(* Logix 5000 project; controller TestController vendor 1 type 14 code 166 rev 32.11; software revision 32.02 *)
// This is a test project

TASK Continuous (continuous, watchdog 500 ms) : MainProgram   // Test continuous task
TASK EventTask (event, rate 10 ms, priority 10, watchdog 500 ms) : EventProgram01   // TestEvent Task
TASK TestTask (periodic, rate 10 ms, priority 10, watchdog 500 ms) : EquipmentPhaseProgram

MODULES
   Local : vendor 1 type 14 code 166 (ICP 0, rev 32.11)
END_MODULES

TYPE AlarmType :   // This is a test alarm type
STRUCT
   DigitalMember : CAM;   // Test digital member
END_STRUCT
END_TYPE

TYPE BoolTest :   // This is a test
STRUCT
   Member01 : BOOL;
   Member02 : BOOL;
   Member04 : BOOL;
   Member05 : BOOL;
END_STRUCT
END_TYPE

TYPE MyStringType :   // This is a test string type
STRUCT
   LEN : DINT;
   DATA : SINT[100];
END_STRUCT
END_TYPE

ADD_ON_INSTRUCTION aoi_Test   (* revision 1.0 *)
// Test AOI
VAR_INPUT
   InputTest : BOOL; {visible}
END_VAR
VAR_OUTPUT
   OutputTest : DINT; {access Read Only, visible}
END_VAR
VAR_IN_OUT
   InOutTest : SimpleType; {constant, required}
END_VAR
VAR_INPUT
   Config : INT; {access None, required}
   Test : BOOL; {access None}
END_VAR
VAR
   LocalBool : BOOL; {access None}
END_VAR

ROUTINE Logic   (* ladder *)
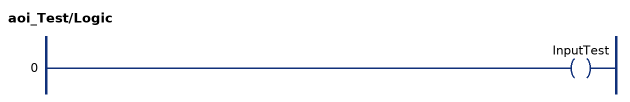
   0: OTE(InputTest);
END_ROUTINE
END_ADD_ON_INSTRUCTION

VAR_GLOBAL   (* controller tags *)
   EquipmentPhaseProgram : PHASE;
   SimpleArray : DINT[10]; {access Read Only}   // This is a test
   SimpleBool : BOOL := 1; {access None}
   SimpleDint : DINT := 3; {access None}
   SimpleInt : INT := 20; {access None}
   SimpleLint : LINT := 3; {access None}
   SimpleReal : REAL; {access None}
   SimpleSint : SINT := 20; {access None}
        .0   // This is a test
   TagParameter : SimpleType; {access None}
   TestAlarmTag : ALARM; {access None}
   TestAnalogAlarm : ALARM_ANALOG;
   TestArrayTypeTag : ArrayType; {access Read Only}
        .SintArray   // Override
   TestComplexTag : ComplexType; {access None}
   TestDigitalAlarm : ALARM_DIGITAL;
   TestStringTag : MyStringType; {access None}
   TestTag01 : SimpleType := (IntMember := 14, DintMember := 1); {access Read Only}
   TestTimer : TIMER := (PRE := 1000); {access None}   // Test Timer
END_VAR

PROGRAM EquipmentPhaseProgram
// Test

ROUTINE Resetting   (* ladder *)
   0: ;
END_ROUTINE

ROUTINE Running   (* ladder *)
END_ROUTINE
END_PROGRAM

PROGRAM EventProgram01   (* main routine Main *)

ROUTINE Main   (* ladder *)
END_ROUTINE
END_PROGRAM

PROGRAM MainProgram   (* main routine Main *)

ROUTINE FBD   (* function block diagram *)
   SHEET 1
END_ROUTINE

ROUTINE Main   (* ladder *)
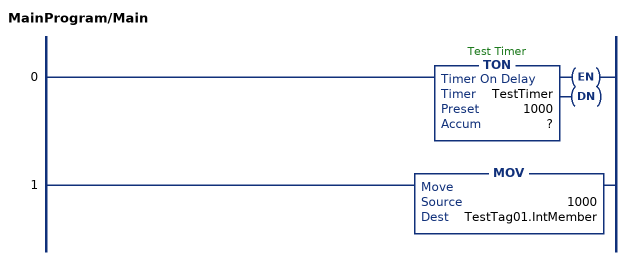
   0: TON(TestTimer,?,?);
   1: MOV(1000,TestTag01.IntMember);
END_ROUTINE

ROUTINE ST   (* structured text *)
   
END_ROUTINE
END_PROGRAM
